// LS Electric XG5000 project: 신호등
// PLC LSPLC

PROGRAM NewProgram (task: 스캔 프로그램)

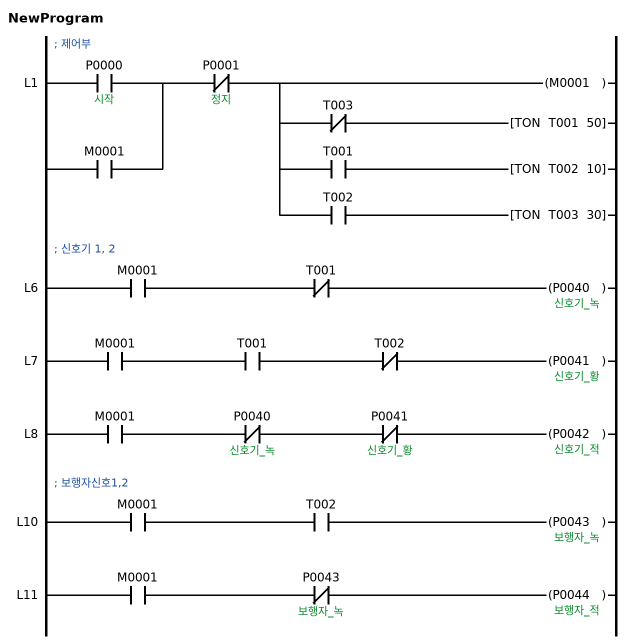
// 제어부
; L1
LOAD      P0000	// 시작
OR        M0001
AND NOT   P0001	// 정지
OUT       M0001
MPUSH
AND NOT   T003
TON       T001 50
MLOAD
AND       T001
TON       T002 10
MPOP
AND       T002
TON       T003 30
// 신호기 1, 2
; L6
LOAD      M0001
AND NOT   T001
OUT       P0040	// 신호기_녹
; L7
LOAD      M0001
AND       T001
AND NOT   T002
OUT       P0041	// 신호기_황
; L8
LOAD      M0001
AND NOT   P0040	// 신호기_녹
AND NOT   P0041	// 신호기_황
OUT       P0042	// 신호기_적
// 보행자신호1,2
; L10
LOAD      M0001
AND       T002
OUT       P0043	// 보행자_녹
; L11
LOAD      M0001
AND NOT   P0043	// 보행자_녹
OUT       P0044	// 보행자_적

VARIABLES AND COMMENTS (devices not used above)
P00002	BIT	점멸